// TwinCAT 3 PLC project Name
// ProgramVersion: 3.1.4026.17
// CompilerDefines: VISU_USEPROPERTYINFO
// libraries:
//   CmpBitmapPool, * (System)
//   Tc2_Standard, * (Beckhoff Automation GmbH)
//   Tc2_System, * (Beckhoff Automation GmbH)
//   Tc2_Utilities, * (Beckhoff Automation GmbH)
//   TextListUtils, * (System)
//   VisuDialogs, * (System)
//   VisuSymbols, 4.5.0.0 (System)
// project tree:
//   DUTs/ DUT_AlarmInfo.TcDUT, DUT_ModelInfo.TcDUT, DUT_ProductData.TcDUT
//   / GlobalTextList.TcGTLO, PlcTask.TcTTO, Visualization Manager.TcVMO (not stored), VISU_TASK.TcTTO
//   GVLs/ GVL_HMI.TcGVL, GVL_Retain.TcGVL, GVL_Status.TcGVL
//   POUs/10_Station/ Station1.TcPOU
//   POUs/70_Data/ Data.TcPOU
//   POUs/80_HMI/ HMI.TcPOU
//   POUs/99_FB/ fbAlarm.TcPOU
//   POUs/ MAIN.TcPOU, Test.TcPOU
//   VISUs/ ImagePool.TcIPO (not stored), TextList.TcTLO
//   VISUs/03_SideFrame/ LowerBar.TcVIS, SideBar.TcVIS, UpperBar.TcVIS
//   VISUs/02_MainFrame/ Main.TcVIS, Data.TcVIS, Alarm.TcVIS, Setting.TcVIS, Manual.TcVIS, Model.TcVIS
//   VISUs/01_Page/ BasePage.TcVIS
// real-time tasks:
//   TASK PlcTask: cycle T#10ms, priority 6, ADS port 351
//   TASK VISU_TASK: cycle T#200000us, priority 8, ADS port 350

CONFIGURATION Name
    RESOURCE PLC ON TwinCAT3
        TASK PlcTask(INTERVAL := T#10ms, PRIORITY := 6);
        TASK VISU_TASK(INTERVAL := T#200000us, PRIORITY := 8);
        PROGRAM MAIN WITH PlcTask : MAIN;
        PROGRAM VisuElems_Visu_Prg WITH VISU_TASK : VisuElems.Visu_Prg;
    END_RESOURCE
END_CONFIGURATION

// ---- DUTs/DUT_AlarmInfo.TcDUT
TYPE DUT_AlarmInfo :
STRUCT
	bActive			: BOOL;              // 알람 활성 여부 (발생 중인지)
	iAlarmCode		: INT;               // 알람 코드 (번호)
	sAlarmMessage	: STRING(255);       // 알람 메시지 텍스트
	tTimeStamp		: DT;                // 알람 발생 시간
	sLocation		: STRING(50);         // 알람 발생 위치 (설비명 등)
	iPriority		: INT;               // 우선순위 (1:높음, 2:중간, 3:낮음 등)
END_STRUCT
END_TYPE

// ---- DUTs/DUT_ModelInfo.TcDUT
TYPE DUT_ModelInfo :
STRUCT
	iNumber		: INT;
	sName		: STRING;
	abType		: ARRAY[1..cMaxTypeNo] OF BOOL;
	aiType		: ARRAY[1..cMaxTypeNo] OF INT;
	arPosition	: ARRAY[1..cMaxPositionNo] OF LREAL;
	arSpeed		: ARRAY[1..cMaxPositionNo] OF LREAL;
END_STRUCT
END_TYPE

// ---- DUTs/DUT_ProductData.TcDUT
TYPE DUT_ProductData :
STRUCT
	sName				:STRING;				(*Product Name*)
	iType				:INT;					(*Product Name*)
	tCycleTime			:TIME;					(*Product Name*)
	tProcessTime		:TIME;					(*Product Name*)
	dtStartTime 		:DT;					(*Product Name*)
	dtEndTime			:DT;					(*Product Name*)
	iRecipeNo			:INT;					(*Product Name*)
	iInputCount			:INT;
	abInspectResult1		:BOOL;	// True = Pass (OK)
	aiInspectResultCode1	:INT;	// 0 = Pending (not inspected yet), 1 = Pass (OK), 2 = Fail – Reason #1, 3 = Fail – Reason #2
	abInspectResult2		:BOOL;	// True = Pass (OK)
	aiInspectResultCode2	:INT;	// 0 = Pending (not inspected yet), 1 = Pass (OK), 2 = Fail – Reason #1, 3 = Fail – Reason #2
	abInspectResult3		:BOOL;	// True = Pass (OK)
	aiInspectResultCode3	:INT;	// 0 = Pending (not inspected yet), 1 = Pass (OK), 2 = Fail – Reason #1, 3 = Fail – Reason #2
	abInspectResult4		:BOOL;	// True = Pass (OK)
	aiInspectResultCode4	:INT;	// 0 = Pending (not inspected yet), 1 = Pass (OK), 2 = Fail – Reason #1, 3 = Fail – Reason #2
	abInspectResult5		:BOOL;	// True = Pass (OK)
	aiInspectResultCode5	:INT;	// 0 = Pending (not inspected yet), 1 = Pass (OK), 2 = Fail – Reason #1, 3 = Fail – Reason #2
	abInspectResult6		:BOOL;	// True = Pass (OK)
	aiInspectResultCode6	:INT;	// 0 = Pending (not inspected yet), 1 = Pass (OK), 2 = Fail – Reason #1, 3 = Fail – Reason #2
END_STRUCT
END_TYPE

// ---- GVLs/GVL_HMI.TcGVL
//{attribute 'qualified_only'}
VAR_GLOBAL
	
	iSelectProductNo	: UINT; // Select Product No.
	bSaveProductData	: BOOL;
	bDeleteProductData	: BOOL;
	bDeleteRecipeData	: BOOL;
	bRemoveProductData	: BOOL;
	
// Main
	bBtAutoMode			: BOOL;
	bBtStart			: BOOL;
	bBtStop				: BOOL;
	bBtHome				: BOOL;
	bBtDoorLock			: BOOL;
	bBtDoorUnlock		: BOOL;
	bBtAlarmReset		: BOOL;
	bLpBlink			: BOOL;
	bLpHome				: BOOL;
	bLpAlarmReset		: BOOL;
	bLpAutoMode			: BOOL;
	bLpStart			: BOOL;
	
// Index
	iTextIndex			: INT;	// By 'TextList' 0= Manual, 1= Auto
	iMainFrame			: INT; // 0= Main, 1= Manual, 2= Setting, 3= Model, 4= Data, 5= Alarm

// Frame Number
    bMainScreen			: BOOL;
    bManualScreen		: BOOL;
	bSettingScreen		: BOOL;
	bModelScreen		: BOOL;
	bDataScreen			: BOOL;
	bAlarmScreen		: BOOL;
	
// Message Box
	sCurrentTitle		: STRING;
	sCurrentMessage		: STRING;
	bCallMessageBox		: BOOL;

// Time
	abStartTimeStamp	: ARRAY[0..cMaxStationNo-1] OF BOOL;
	abEndTimeStamp		: ARRAY[0..cMaxStationNo-1] OF BOOL;
	sCurrentTime		: STRING;

// Model
	iInputModelNo		: INT;
	bBtSaveModelData	: BOOL;
	bLpSaveModelData	: BOOL;
	bBtActivateModel	: BOOL;
	bLpActivateModel	: BOOL;
	bLpDiffNumber		: BOOL;
	bLpDiffName			: BOOL;
	bLpDiffbType		: BOOL;
	bLpDiffiType		: BOOL;
	bLpDiffrPosition	: BOOL;
	bLpDiffrSpeed		: BOOL;
	iModelIndex			: INT := 1;
	bInvisibleLeft		: BOOL;
	bInvisibleRight		: BOOL;

// Test Bt
	bTest				: BOOL;
END_VAR

// ---- GVLs/GVL_Retain.TcGVL
//{attribute 'qualified_only'}
 {attribute 'TcPersistent'}
VAR_GLOBAL PERSISTENT
//Product Data
	astProductData 		: ARRAY[0..cMaxStationNo+1] OF DUT_ProductData;
	abMoveShift			: ARRAY[0..cMaxStationNo] OF BOOL;

// Alarm
	astAlarmHistory		: ARRAY[0..cMaxAlarmLogCount-1] OF DUT_AlarmInfo; // 최근 100개 알람 저장

// Model
	astInputModel		: ARRAY[1..cMaxModelNo] OF dut_ModelInfo;
	astModel			: ARRAY[1..cMaxModelNo] OF dut_ModelInfo;
	stCurrnetModel		: dut_ModelInfo;	
END_VAR

VAR_GLOBAL CONSTANT
	cMaxAlarmLogCount	: INT := 100; 
	cMaxStationNo 		: INT := 30;
	cMaxTypeNo			: INT := 20;
	cMaxPositionNo		: INT := 30;
	cMaxModelNo			: INT := 10;
	cMaxStationAlarmNo	: INT := 100;
	
END_VAR

// ---- GVLs/GVL_Status.TcGVL
//{attribute 'qualified_only'}
VAR_GLOBAL
	//DataShift
		fbLocalTime 		: FB_LocalSystemTime;
		
	//Status
		bAutoMode				:BOOL;
		bManualMode				:BOOL;
		bHomeMode				:BOOL;
		bAutoBusy				:BOOL;
		bHomeBusy				:BOOL;
		bManualBusy				:BOOL;
		bAlarm					:BOOL;
		bWarning				:BOOL;
		bHomeComplete			:BOOL;
		bSafetyDoorLocked		:BOOL;
		bSafetyDoorUnlocked		:BOOL;
		bAlarmReset				: BOOL;
		
	//Command
		bStopCmd		:BOOL;
		bAutoCmd		:BOOL;
		bHomeCmd		:BOOL;
		bDoorUnlockCmd	:BOOL;
		bDoorLockCmd	:BOOL;
		
END_VAR

// ---- POUs/MAIN.TcPOU
PROGRAM MAIN
VAR
	
END_VAR

Data();
HMI();
Station1();

IF GVL_HMI.bTest THEN
	Test();	
END_IF

END_PROGRAM

// ---- POUs/70_Data/Data.TcPOU
PROGRAM Data
VAR
	i					:INT; //loop index
END_VAR

// Local Time
	GVL_Status.fbLocalTime(bEnable := TRUE);	// Current Time

//Remove Total Product Data
	IF GVL_HMI.bRemoveProductData THEN
		FOR i := 0 TO cMaxStationNo DO
			astProductData[i] := astProductData[cMaxStationNo+1];
		END_FOR;
		GVL_HMI.bRemoveProductData := FALSE;
	END_IF

//Data Shift
	FOR i := 0 TO (cMaxStationNo) DO
		IF i > 0 AND i <= cMaxStationNo THEN  // 범위 체크 추가
			IF abMoveShift[i] = TRUE THEN
				astProductData[i] := astProductData[i-1];
				astProductData[i-1] := astProductData[cMaxStationNo+1]; // Delete Data before Station
				abMoveShift[i] := FALSE;
			END_IF
			
			IF abStartTimeStamp[i] AND GVL_Status.fbLocalTime.bValid THEN
				astProductData[i].dtStartTime := SYSTEMTIME_TO_DT(GVL_Status.fbLocalTime.systemTime);
			END_IF
			IF abEndTimeStamp[i] AND GVL_Status.fbLocalTime.bValid THEN
				astProductData[i].dtEndTime := SYSTEMTIME_TO_DT(GVL_Status.fbLocalTime.systemTime);
			END_IF		
			astProductData[i].tProcessTime	:= astProductData[i].dtEndTime - astProductData[i].dtStartTime;
		END_IF
	END_FOR;

END_PROGRAM

// ---- POUs/80_HMI/HMI.TcPOU
PROGRAM HMI
VAR
	tonBlink : ton;
	tonAlarmReset : ton;
	i	: INT;
	iDiffReset: INT;
	triModelSet: R_TRIG;
END_VAR

// Current Time
	GVL_HMI.sCurrentTime := SYSTEMTIME_TO_STRING( GVL_Status.fbLocalTime.systemTime);

// Select Auto Mode
	IF GVL_Status.bAutoCmd = FALSE AND GVL_Status.bAutoBusy = FALSE AND GVL_Status.bManualBusy = FALSE AND GVL_Status.bHomeBusy = FALSE  THEN
		//Turn On Auto Mode 
        IF GVL_HMI.bBtAutoMode = TRUE AND GVL_Status.bAutoMode = FALSE AND GVL_Status.bSafetyDoorLocked THEN
			GVL_Status.bAutoMode := TRUE;
			GVL_HMI.bBtAutoMode := FALSE;
		END_IF
		//Turn Off Auto Mode
		IF GVL_HMI.bBtAutoMode = TRUE AND GVL_Status.bAutoMode = TRUE  THEN
			GVL_Status.bAutoMode := FALSE;
			GVL_HMI.bBtAutoMode := FALSE;
		END_IF
	ELSE
		GVL_HMI.bBtAutoMode := FALSE;
	END_IF
		
        IF GVL_Status.bSafetyDoorUnlocked OR (NOT bDoorUnlockCmd AND NOT bDoorLockCmd)  THEN
		GVL_HMI.bBtAutoMode := FALSE;
	END_IF
	
	gvl_hmi.bLpAutoMode := GVL_Status.bAutoMode OR ( GVL_HMI.bLpBlink AND GVL_Status.bHomeComplete AND GVL_Status.bHomeMode);
	
// Select Manual Mode
	IF GVL_Status.bAutoMode = FALSE THEN
		GVL_Status.bManualMode := TRUE;
		GVL_HMI.iTextIndex := 0;
	ELSE
		GVL_Status.bManualMode := FALSE;
		GVL_HMI.iTextIndex := 1;
	END_IF
	
// Auto Running
	IF GVL_HMI.bBtStart = TRUE AND GVL_Status.bAutoMode = TRUE AND GVL_Status.bHomeComplete = TRUE AND GVL_Status.bAutoBusy = FALSE AND GVL_Status.bManualBusy = FALSE AND GVL_Status.bHomeBusy = FALSE THEN
		GVL_Status.bAutoCmd := TRUE;
		GVL_HMI.bBtStart := FALSE;
	ELSIF GVL_HMI.bBtStart = TRUE AND GVL_Status.bAutoMode = FALSE THEN
		GVL_HMI.bBtStart := FALSE;
	END_IF
	
	gvl_hmi.bLpStart := GVL_Status.bAutoCmd OR ( GVL_HMI.bLpBlink AND GVL_Status.bHomeComplete AND GVL_Status.bAutoMode AND ( NOT gvl_status.bAlarm AND NOT gvl_status.bWarning));
	
	
// Stop 
	IF GVL_HMI.bBtStop = TRUE AND GVL_Status.bStopCmd = FALSE THEN
		GVL_Status.bStopCmd	:= TRUE;
		GVL_HMI.bBtStop := FALSE;
	END_IF
	
	IF GVL_Status.bStopCmd = TRUE AND GVL_Status.bAutoBusy = FALSE AND GVL_Status.bManualBusy = FALSE AND GVL_Status.bHomeBusy = FALSE THEN
		GVL_Status.bAutoCmd := FALSE;
		GVL_Status.bHomeCmd := FALSE;
		GVL_Status.bStopCmd := FALSE;
		GVL_HMI.bBtStop := FALSE;
	END_IF
	
// Home 
	GVL_Status.bHomeMode := GVL_Status.bSafetyDoorLocked AND GVL_Status.bManualMode;
	
	IF GVL_HMI.bBtHome = TRUE AND GVL_Status.bHomeMode = TRUE AND GVL_Status.bAutoBusy = FALSE AND GVL_Status.bManualBusy = FALSE AND GVL_Status.bHomeBusy = FALSE AND GVL_Status.bAutoCmd = FALSE THEN
		GVL_Status.bHomeCmd := TRUE;
		GVL_HMI.bBtHome := FALSE;
	ELSIF GVL_HMI.bBtHome = TRUE AND GVL_Status.bHomeMode = FALSE THEN
		GVL_HMI.bBtHome := FALSE;
	END_IF
	
	IF GVL_Status.bHomeCmd = TRUE AND GVL_Status.bHomeComplete = TRUE THEN
		GVL_Status.bHomeCmd := FALSE;
	END_IF
	
	// bHomeComplete Reset
		IF GVL_Status.bSafetyDoorUnlocked THEN
			GVL_Status.bHomeComplete := FALSE;
		END_IF
	
		GVL_HMI.bLpHome := GVL_Status.bHomeComplete OR ( NOT GVL_Status.bHomeComplete AND GVL_Status.bHomeMode AND GVL_HMI.bLpBlink);
	
// Door Unlock
	IF GVL_HMI.bBtDoorUnlock AND GVL_Status.bManualMode AND NOT GVL_Status.bManualBusy THEN
		GVL_Status.bDoorUnlockCmd := TRUE;
		GVL_Status.bDoorLockCmd := FALSE;
		GVL_HMI.bBtDoorUnlock := FALSE;
	ELSE
		GVL_HMI.bBtDoorUnlock := FALSE;
	END_IF
	
// Door Lock
	IF GVL_HMI.bBtDoorLock AND GVL_Status.bManualMode AND NOT GVL_Status.bManualBusy THEN
		GVL_Status.bDoorLockCmd := TRUE;
		GVL_Status.bDoorUnlockCmd := FALSE;
		GVL_HMI.bBtDoorLock := FALSE;
	ELSE
		GVL_HMI.bBtDoorLock := FALSE;
	END_IF
	
// Alarm Reset
	IF gvl_hmi.bBtAlarmReset THEN
		GVL_Status.bAlarmReset := TRUE;
		gvl_hmi.bBtAlarmReset := FALSE;
	END_IF
	
	tonAlarmReset(in := GVL_Status.bAlarmReset, pt := T#0.5S);
	
	IF tonAlarmReset.Q THEN
		GVL_Status.bAlarmReset := FALSE;
	END_IF
	
	gvl_hmi.bLpAlarmReset := GVL_Status.bAlarmReset OR (GVL_HMI.bLpBlink AND (gvl_status.bAlarm OR gvl_status.bWarning));
		
// blink
 	tonBlink(in := NOT tonBlink.q , PT := T#500MS);
	
	IF tonBlink.Q THEN
		GVL_HMI.bLpBlink := NOT GVL_HMI.bLpBlink;
	END_IF
	
// Current Screen
	gvl_hmi.bMainScreen := gvl_hmi.iMainFrame = 0;
	gvl_hmi.bManualScreen := gvl_hmi.iMainFrame = 1;
	gvl_hmi.bSettingScreen := gvl_hmi.iMainFrame = 2;
	gvl_hmi.bModelScreen := gvl_hmi.iMainFrame = 3;
	gvl_hmi.bDataScreen := gvl_hmi.iMainFrame = 4;
	gvl_hmi.bAlarmScreen := gvl_hmi.iMainFrame = 5;
	
	
// Model
	 IF bModelScreen THEN
		 FOR i := 1 TO cMaxModelNo DO
			astInputModel[i].iNumber := i;
			IF bBtSaveModelData THEN
				astModel[iModelindex] := astInputModel[iModelindex];
			END_IF
			IF bBtActivateModel THEN
				 stCurrnetModel := astModel[iModelindex];
			END_IF
		 END_FOR
		 iModelindex := LIMIT(1,iModelindex,cMaxModelNo);
		 bLpDiffNumber := astInputModel[iModelindex].iNumber <> astModel[iModelindex].iNumber;
		 bLpDiffName := astInputModel[iModelindex].sName <> astModel[iModelindex].sName;
		 FOR i := 1 TO cMaxTypeNo DO
			 IF astInputModel[iModelindex].abType[i] <> astModel[iModelindex].abType[i] THEN
			 bLpDiffbType := TRUE;
			 END_IF
		 END_FOR
		 FOR i := 1 TO cMaxTypeNo DO
			 IF astInputModel[iModelindex].aiType[i] <> astModel[iModelindex].aiType[i] THEN
			 bLpDiffiType := TRUE;
			 END_IF
		 END_FOR
		 FOR i := 1 TO cMaxPositionNo DO
			 IF astInputModel[iModelindex].arPosition[i] <> astModel[iModelindex].arPosition[i] THEN
			 bLpDiffrPosition := TRUE;
			 END_IF
		 END_FOR
		 FOR i := 1 TO cMaxPositionNo DO
			 IF astInputModel[iModelindex].arSpeed[i] <> astModel[iModelindex].arSpeed[i] THEN
			 bLpDiffrSpeed := TRUE;
			 END_IF
		 END_FOR		
		 IF (iModelindex <> iDiffReset) OR bBtSaveModelData OR triModelSet.Q THEN
			 bLpDiffbType := FALSE;
			 bLpDiffiType := FALSE;
			 bLpDiffrPosition := FALSE;
			 bLpDiffrSpeed := FALSE;
			 iDiffReset := iModelindex;
		 END_IF
		 bLpSaveModelData := bBtSaveModelData OR ((bLpDiffNumber OR bLpDiffName OR bLpDiffbType OR bLpDiffiType OR bLpDiffrPosition OR bLpDiffrSpeed) AND bLpBlink);
		 bInvisibleLeft := iModelindex = 1;
		 bInvisibleRight := iModelindex = cMaxModelNo;
		 bLpActivateModel := ((NOT bLpSaveModelData AND (stCurrnetModel.iNumber = 0)) AND bLpBlink) OR bBtActivateModel;
	 END_IF
	 triModelSet(CLK:= bModelScreen, Q=> );
	 IF triModelSet.Q THEN
		 FOR i := 1 TO cMaxModelNo DO
			astInputModel[i] := astModel[i];
		 END_FOR
	 END_IF

END_PROGRAM

// ---- POUs/10_Station/Station1.TcPOU
PROGRAM Station1
VAR

END_VAR

END_PROGRAM

// ---- POUs/Test.TcPOU
PROGRAM Test
VAR

	fbTestAlarm1: fbalarm;

        bTestSelectWarning: BOOL;
        bTestAlarmCondition: BOOL;
	bTestError1: BOOL;
	bTestWarning1: BOOL;
	

END_VAR

// Door		
	GVL_Status.bSafetyDoorLocked := GVL_Status.bDoorLockCmd;
	GVL_Status.bSafetyDoorUnlocked := GVL_Status.bDoorUnlockCmd;
	
// home
	IF GVL_Status.bHomeCmd THEN
		GVL_Status.bHomeComplete := TRUE;
	END_IF



// Alarm
	fbTestAlarm1(
        bSelectWarning:= bTestSelectWarning,
	tDelayTime:= T#1S, 
	bCommand:= TRUE, 
        bAlarmCondition:= bTestAlarmCondition,
	iAlarmCode:= 1, 
	iPriority:= 1, 
	sAlarmMessage:= 'hello', 
	sLocation:= 'office', 
	bError=> bTestError1, 
	bWarning=> bTestWarning1);

END_PROGRAM

// ---- POUs/99_FB/fbAlarm.TcPOU
FUNCTION_BLOCK fbAlarm	// 
VAR_INPUT
	bSelectWarning	: BOOL;
	tDelayTime	: TIME;
	bCommand	: BOOL;
	bAlarmCondition	: BOOL;
	iAlarmCode	: INT;
	iPriority	: INT;
	sAlarmMessage	: STRING;
	sLocation	: STRING;
END_VAR
VAR_OUTPUT
	bError	: BOOL;
	bWarning	: BOOL;
END_VAR
VAR
	bAlarm	: BOOL;
	triAlarm	: R_Trig;
	triWarning	: R_Trig;
	triError	: R_Trig;
	i: INT;
	stAlarmInfo	: Dut_AlarmInfo;
	tonDelayTimer	: ton;
END_VAR


// Alarm Input
	bAlarm	:= bCommand AND bAlarmCondition;
	tonDelayTimer(in := bAlarm, pt :=tDelayTime);

// Alarm History
	triAlarm(clk := tonDelayTimer.Q);
	IF triAlarm.Q THEN
		FOR i := cMaxAlarmLogCount TO 1 BY -1 DO
			astAlarmHistory[i]	:= astAlarmHistory[i-1];
		END_FOR
		stAlarmInfo.iAlarmCode	:= iAlarmCode;
		stAlarmInfo.iPriority	:= iPriority;
		stAlarmInfo.sAlarmMessage	:= sAlarmMessage;
		stAlarmInfo.sLocation	:= sLocation;
		stAlarmInfo.tTimeStamp	:= SYSTEMTIME_TO_DT(GVL_Status.fbLocalTime.systemTime);
		astAlarmHistory[0] := stAlarmInfo;
	END_IF

// Alarm Output
	IF tonDelayTimer.Q THEN
		bError := NOT bSelectWarning;
		gvl_status.bAlarm := NOT bSelectWarning;
		bWarning := bSelectWarning;
		gvl_status.bWarning := bSelectWarning;
	END_IF
	
// Alarm Reset
	IF bAlarmReset THEN
		bError := FALSE;
		bWarning := FALSE;
		gvl_status.bAlarm := FALSE;
		gvl_status.bWarning := FALSE;
	END_IF
	
// Call Message Box
	triWarning(clk := gvl_status.bWarning);
	IF triWarning.Q THEN
		sCurrentTitle	:= astAlarmHistory[0].sLocation;
		sCurrentMessage	:= astAlarmHistory[0].sAlarmMessage;
		bCallMessageBox := gvl_status.bWarning;
	END_IF
	
// Change Main Frame to Alarm
	triError(clk := gvl_status.bAlarm);
	IF triError.Q THEN
		iMainFrame := 5;
	END_IF

END_FUNCTION_BLOCK

// ---- GlobalTextList.TcGTLO
TEXTLIST GlobalTextList
  422 = '%.19s' | Korea: '%.19s' | English: '%.19s'
  792 = '%i'
  75 = '%s'
  500 = '1'
  410 = 'a'
  336 = 'Activate Model'
  479 = 'Activate Name : %s'
  578 = 'Activate No : %i'
  851 = 'Active'
  609 = 'Alarm'
  662 = 'Alarm Code'
  947 = 'Alarm Page'
  35 = 'Alarm Reset'
  411 = 'AlarmCode'
  22 = 'AlarmMessage'
  147 = 'AlarmReset' | Korea: '초기화'
  23 = 'Alarm_Log'
  557 = 'Arkplus' | Korea: '화면인터페이스' | English: 'Standard_HMI'
  984 = 'Assemble1'
  741 = 'Assemble2'
  530 = 'Assemble3'
  491 = 'Auto Mode'
  808 = 'AutoMode'
  787 = 'b'
  699 = 'Code'
  709 = 'Conveyor'
  734 = 'Conveyor Pitch'
  977 = 'Current %s'
  122 = 'Data'
  161 = 'Data Page'
  928 = 'dfasdffffffffffffffffffffffffffffff'
  215 = 'Disable'
  226 = 'Door'
  850 = 'Door Close'
  103 = 'Door Open'
  567 = 'DoorClose'
  32 = 'Enable'
  271 = 'English' | Korea: '영어' | English: 'English'
  697 = 'fdsafdafsda'
  217 = 'GroupBox'
  279 = 'Home'
  993 = 'Inspection1'
  456 = 'Inspection2'
  921 = 'Inspection3'
  332 = 'Korea' | Korea: '한국어' | English: 'Korea'
  0 = 'Location'
  956 = 'Main'
  707 = 'Main Page'
  301 = 'Manual'
  775 = 'Manual Page'
  83 = 'ManualMode'
  186 = 'Message'
  376 = 'Model'
  601 = 'Model Name %s'
  313 = 'Model Page'
  136 = 'Name'
  599 = 'Name %s'
  828 = 'No : %i'
  259 = 'No : %s'
  536 = 'Parameter'
  975 = 'Pos %5.2f'
  395 = 'Pos %d'
  403 = 'Priority'
  529 = 'Robot'
  204 = 'SafetyBypass'
  331 = 'Sample'
  908 = 'Save Model'
  239 = 'Setting'
  394 = 'Setting Page'
  181 = 'Spd %5.2f'
  125 = 'Speed'
  849 = 'Standard_HMI' | Korea: '화면인터페이스'
  261 = 'Start'
  606 = 'Stop'
  904 = 'Test'
  272 = 'Time Stamp'
  199 = 'TimeStamp'
  396 = 'TurnTable'
  712 = 'type'
  334 = 'Type01'
  446 = 'Type02'
  966 = 'Type03'
  706 = 'Type04'
  126 = 'Type05'
  809 = 'Type06'
  245 = 'Type07'
  162 = 'Type08'
  992 = 'Type09'
  710 = 'Type10'
  26 = 'Unit1 Assemble'
  926 = 'Unit1 End'
  600 = 'Unit1 Position1'
  943 = 'Unit1 Start'
  540 = 'Unit2 Position1'
  942 = 'Unit2 Start'
  16 = 'Unit3 Assemble'
  358 = 'Unit3 End'
  93 = 'Vision'
  773 = 'Vision1'
  925 = 'Vision2'
  185 = 'Vision3'
  171 = 'yyyy‑MM‑dd\xa0HH:mm:ss'
END_TEXTLIST

// ---- VISUs/03_SideFrame/LowerBar.TcVIS
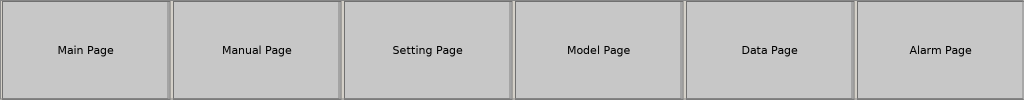
VISUALIZATION LowerBar  // 1024x100
    Button (2,1 168x99), "Main Page", colour toggle: gvl_hmi.bMainScreen
        OnMouseClick: execute { gvl_hmi.iMainFrame := 0; }
    Button (173,1 168x99), "Manual Page", colour toggle: gvl_hmi.bManualScreen
        OnMouseClick: execute { gvl_hmi.iMainFrame := 1; }
    Button (344,1 168x99), "Setting Page", colour toggle: gvl_hmi.bSettingScreen
        OnMouseClick: execute { gvl_hmi.iMainFrame := 2; }
    Button (515,1 168x99), "Model Page", colour toggle: gvl_hmi.bModelScreen
        OnMouseClick: execute { gvl_hmi.iMainFrame := 3; }
    Button (686,1 168x99), "Data Page", colour toggle: gvl_hmi.bDataScreen
        OnMouseClick: execute { gvl_hmi.iMainFrame := 4; }
    Button (857,1 168x99), "Alarm Page", colour toggle: gvl_hmi.bAlarmScreen
        OnMouseClick: execute { gvl_hmi.iMainFrame := 5; }
END_VISUALIZATION

// ---- VISUs/03_SideFrame/SideBar.TcVIS
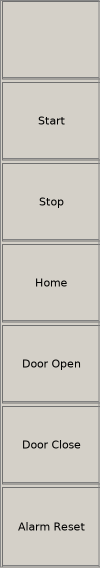
VISUALIZATION SideBar  // 100x568
    Button (2,1 99x78), colour toggle: GVL_HMI.bLpAutoMode, text list: 'TextList', text index: GVL_HMI.iTextIndex
        OnMouseClick: execute { GVL_HMI.bBtAutoMode := true; }
    Button (2,82 99x78), "Start", colour toggle: gvl_hmi.bLpStart
        OnMouseClick: execute { GVL_HMI.bBtStart := TRUE; }
    Button (2,163 99x78), "Stop", colour toggle: GVL_Status.bStopCmd
        OnMouseClick: execute { GVL_HMI.bBtStop := True; }
    Button (2,244 99x78), "Home", colour toggle: GVL_HMI.bLpHome
        OnMouseClick: execute { GVL_HMI.bBtHome := True; }
    Button (2,325 99x78), "Door Open", colour toggle: GVL_Status.bSafetyDoorUnlocked
        OnMouseClick: execute { GVL_HMI.bBtDoorUnlock := True; }
    Button (2,406 99x78), "Door Close", colour toggle: GVL_Status.bSafetyDoorLocked
        OnMouseClick: execute { GVL_HMI.bBtDoorLock := True; }
    Button (2,487 99x80), "Alarm Reset", colour toggle: gvl_hmi.bLpAlarmReset
        OnMouseClick: execute { GVL_HMI.bBtAlarmReset := True; }
END_VISUALIZATION

// ---- VISUs/03_SideFrame/UpperBar.TcVIS
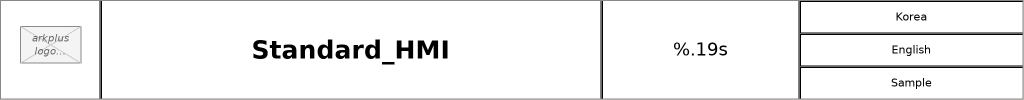
VISUALIZATION UpperBar  // 1024x100
    Rectangle (0,0 100x99)
    Image (20,26 61x37), image: arkplus logo_Resize
    Rectangle (101,0 500x99), "Standard_HMI"
    Rectangle (602,0 197x99), "%.19s", text variable: GVL_HMI.sCurrentTime
    Rectangle (800,1 223x32), "Korea"
        OnMouseClick: ChangeLanguage ChangeLanguage=Korea
    Rectangle (800,34 223x32), "English"
        OnMouseClick: ChangeLanguage ChangeLanguage=English
    Rectangle (800,67 223x32), "Sample"
END_VISUALIZATION

// ---- VISUs/02_MainFrame/Main.TcVIS
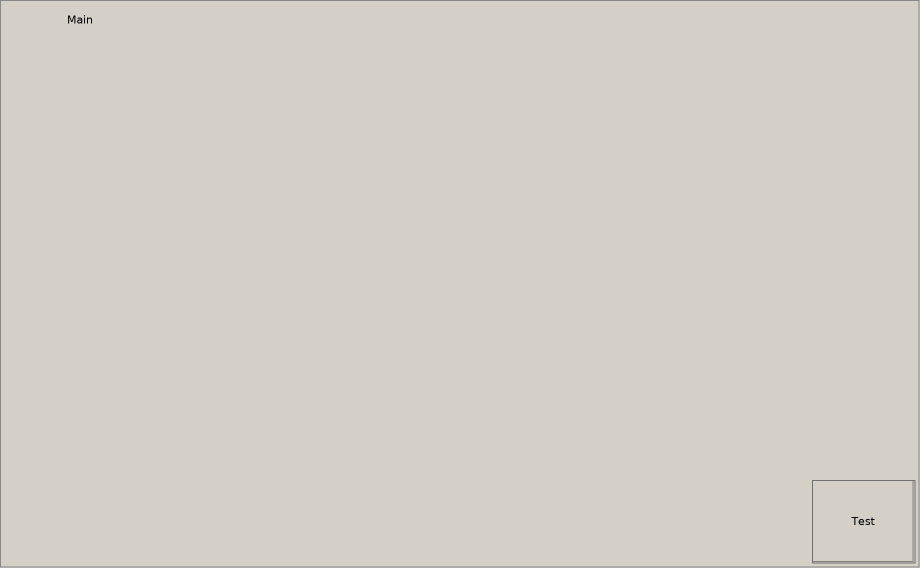
VISUALIZATION Main  // 920x568
    Label (5,5 150x30), "Main"
    Button (812,480 103x83), "Test", colour toggle: GVL_HMI.bTest
        toggle GVL_HMI.bTest
END_VISUALIZATION

// ---- VISUs/02_MainFrame/Data.TcVIS
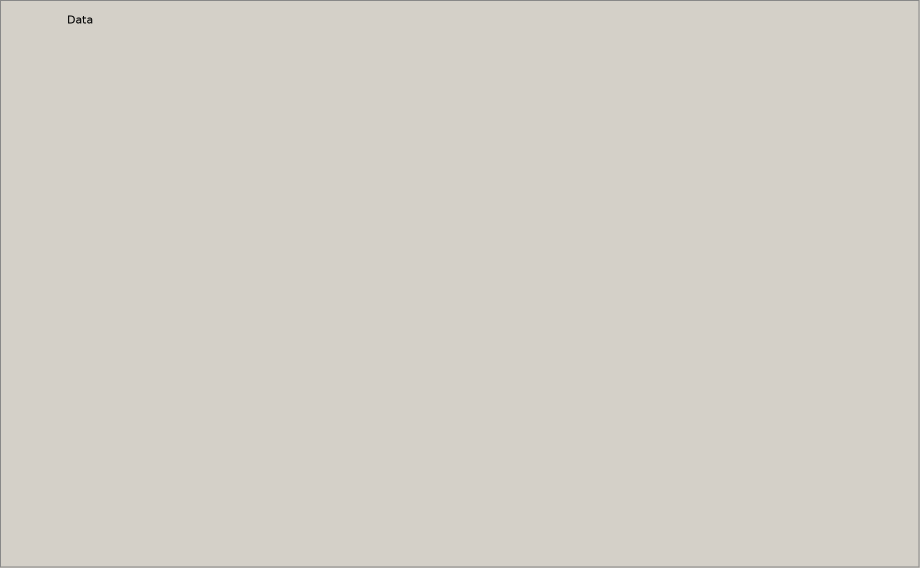
VISUALIZATION Data  // 920x568
    Label (5,5 150x30), "Data"
END_VISUALIZATION

// ---- VISUs/02_MainFrame/Alarm.TcVIS
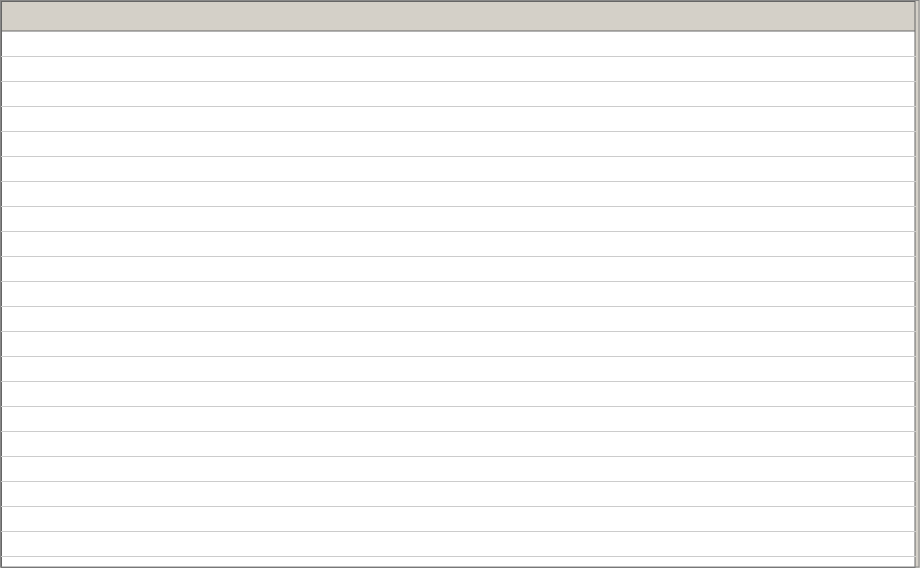
VISUALIZATION Alarm  // 920x568
    Table (1,1 914x567), data array: GVL_Retain.astAlarmHistory
        p3854506369: GVL_Retain.astAlarmHistory[INDEX].bActive
        p1892666644: GVL_Retain.astAlarmHistory[INDEX].iAlarmCode
        p338671338: GVL_Retain.astAlarmHistory[INDEX].sAlarmMessage
        p2170511999: GVL_Retain.astAlarmHistory[INDEX].tTimeStamp
        p3723444502: GVL_Retain.astAlarmHistory[INDEX].sLocation
        p1218418051: GVL_Retain.astAlarmHistory[INDEX].iPriority
        p4092479075: Time Stamp
        p1014161805: 99 - 0 + INT#1
        p1128707560: cMaxAlarmLogCount
END_VISUALIZATION

// ---- VISUs/02_MainFrame/Setting.TcVIS
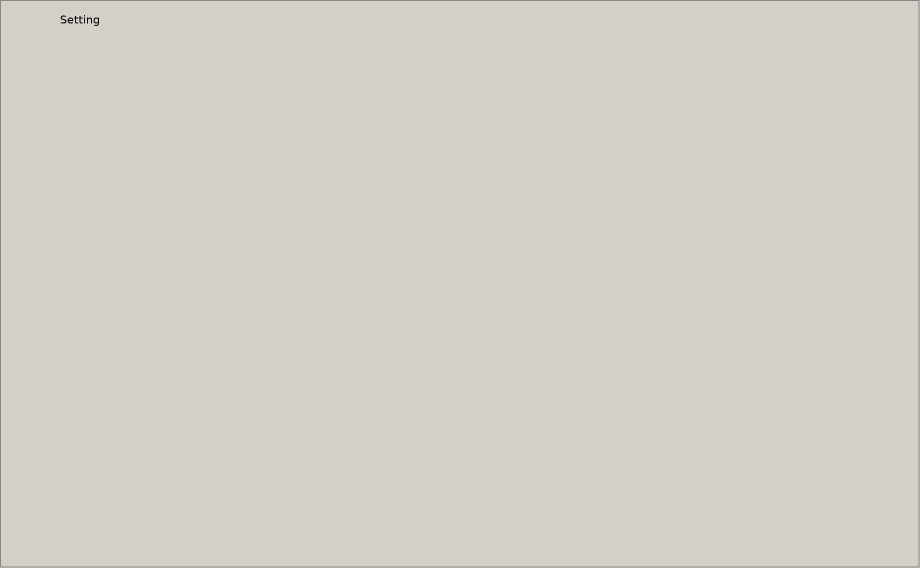
VISUALIZATION Setting  // 920x568
    Label (5,5 150x30), "Setting"
END_VISUALIZATION

// ---- VISUs/02_MainFrame/Manual.TcVIS
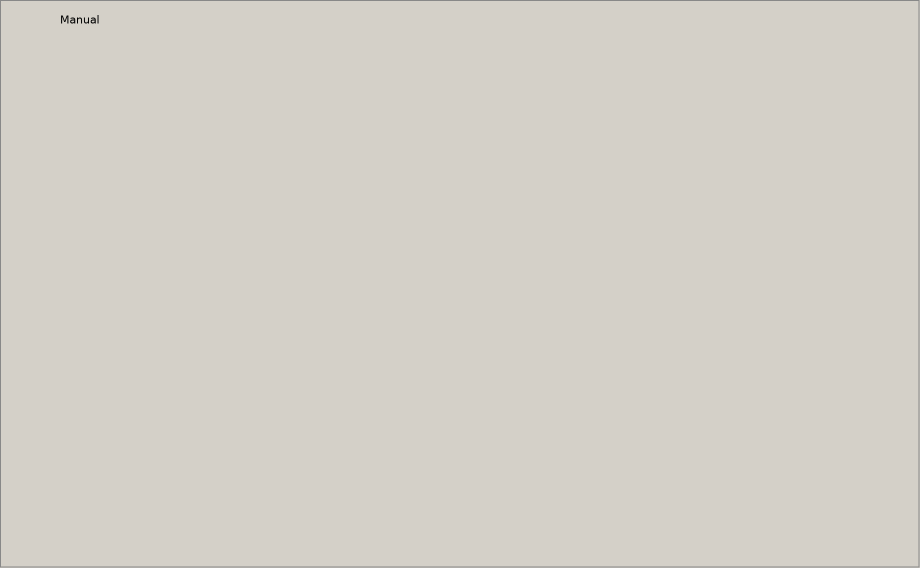
VISUALIZATION Manual  // 920x568
    Label (5,5 150x30), "Manual"
END_VISUALIZATION

// ---- VISUs/02_MainFrame/Model.TcVIS
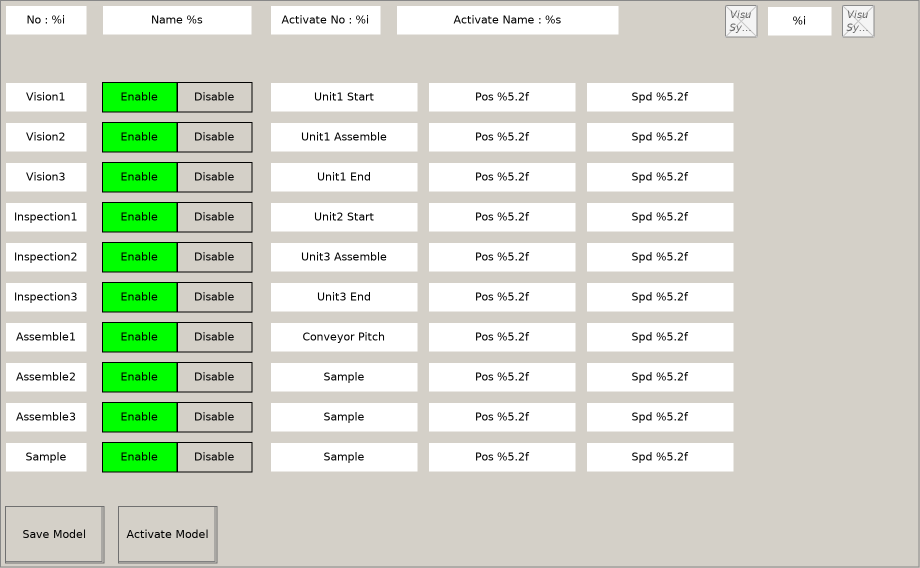
VISUALIZATION Model  // 920x568
    Textfield (102,5 150x30), "Name %s", text variable: astInputModel[iModelIndex].sName
        OnMouseClick: write the text variable via Edit
    Textfield (5,5 82x30), "No : %i", text variable: astInputModel[iModelIndex].iNumber
    Image (725,5 32x32), invisible if: bInvisibleLeft, image: VisuSymbols.Symbols.ArrowBoldLeft
        OnMouseClick: execute { iModelindex := iModelindex -1; }
    Image (842,5 32x32), invisible if: bInvisibleRight, image: VisuSymbols.Symbols.ArrowBoldRight
        OnMouseClick: execute { iModelindex := iModelindex +1; }
    Textfield (767,6 65x30), "%i", text variable: astInputModel[iModelIndex].iNumber
        OnMouseClick: write iModelIndex via Default, min 1, max cMaxModelNo
    Textfield (5,82 82x30), "Vision1"
    Rectangle (102,82 75x30), "Enable", colour toggle: astInputModel[iModelIndex].abType[1]
        OnMouseClick: execute { astInputModel[iModelIndex].abType[1] := FALSE; }
    Rectangle (177,82 75x30), "Disable", colour toggle: astInputModel[iModelIndex].abType[1]
        OnMouseClick: execute { astInputModel[iModelIndex].abType[1] := true; }
    Textfield (5,122 82x30), "Vision2"
    Rectangle (102,122 75x30), "Enable", colour toggle: astInputModel[iModelIndex].abType[2]
        OnMouseClick: execute { astInputModel[iModelIndex].abType[2] := FALSE; }
    Rectangle (177,122 75x30), "Disable", colour toggle: astInputModel[iModelIndex].abType[2]
        OnMouseClick: execute { astInputModel[iModelIndex].abType[2] := true; }
    Textfield (5,162 82x30), "Vision3"
    Rectangle (102,162 75x30), "Enable", colour toggle: astInputModel[iModelIndex].abType[3]
        OnMouseClick: execute { astInputModel[iModelIndex].abType[3] := FALSE; }
    Rectangle (177,162 75x30), "Disable", colour toggle: astInputModel[iModelIndex].abType[3]
        OnMouseClick: execute { astInputModel[iModelIndex].abType[3] := true; }
    Textfield (5,202 82x30), "Inspection1"
    Rectangle (102,202 75x30), "Enable", colour toggle: astInputModel[iModelIndex].abType[4]
        OnMouseClick: execute { astInputModel[iModelIndex].abType[4] := FALSE; }
    Rectangle (177,202 75x30), "Disable", colour toggle: astInputModel[iModelIndex].abType[4]
        OnMouseClick: execute { astInputModel[iModelIndex].abType[4] := true; }
    Textfield (5,242 82x30), "Inspection2"
    Rectangle (102,242 75x30), "Enable", colour toggle: astInputModel[iModelIndex].abType[5]
        OnMouseClick: execute { astInputModel[iModelIndex].abType[5] := FALSE; }
    Rectangle (177,242 75x30), "Disable", colour toggle: astInputModel[iModelIndex].abType[5]
        OnMouseClick: execute { astInputModel[iModelIndex].abType[5] := true; }
    Textfield (5,282 82x30), "Inspection3"
    Rectangle (102,282 75x30), "Enable", colour toggle: astInputModel[iModelIndex].abType[6]
        OnMouseClick: execute { astInputModel[iModelIndex].abType[6] := FALSE; }
    Rectangle (177,282 75x30), "Disable", colour toggle: astInputModel[iModelIndex].abType[6]
        OnMouseClick: execute { astInputModel[iModelIndex].abType[6] := true; }
    Textfield (5,322 82x30), "Assemble1"
    Rectangle (102,322 75x30), "Enable", colour toggle: astInputModel[iModelIndex].abType[7]
        OnMouseClick: execute { astInputModel[iModelIndex].abType[7] := FALSE; }
    Rectangle (177,322 75x30), "Disable", colour toggle: astInputModel[iModelIndex].abType[7]
        OnMouseClick: execute { astInputModel[iModelIndex].abType[7] := true; }
    Textfield (5,362 82x30), "Assemble2"
    Rectangle (102,362 75x30), "Enable", colour toggle: astInputModel[iModelIndex].abType[8]
        OnMouseClick: execute { astInputModel[iModelIndex].abType[8] := FALSE; }
    Rectangle (177,362 75x30), "Disable", colour toggle: astInputModel[iModelIndex].abType[8]
        OnMouseClick: execute { astInputModel[iModelIndex].abType[8] := true; }
    Textfield (5,402 82x30), "Assemble3"
    Rectangle (102,402 75x30), "Enable", colour toggle: astInputModel[iModelIndex].abType[9]
        OnMouseClick: execute { astInputModel[iModelIndex].abType[9] := FALSE; }
    Rectangle (177,402 75x30), "Disable", colour toggle: astInputModel[iModelIndex].abType[9]
        OnMouseClick: execute { astInputModel[iModelIndex].abType[9] := true; }
    Textfield (5,442 82x30), "Sample"
    Rectangle (102,442 75x30), "Enable", colour toggle: astInputModel[iModelIndex].abType[10]
        OnMouseClick: execute { astInputModel[iModelIndex].abType[10] := FALSE; }
    Rectangle (177,442 75x30), "Disable", colour toggle: astInputModel[iModelIndex].abType[10]
        OnMouseClick: execute { astInputModel[iModelIndex].abType[10] := true; }
    Button (5,506 99x57), "Save Model", colour toggle: bLpSaveModelData
        tap bBtSaveModelData
    Button (118,506 99x57), "Activate Model", colour toggle: bLpActivateModel
        tap bBtActivateModel
    Textfield (396,5 223x30), "Activate Name : %s", text variable: stCurrnetModel.sName
        OnMouseClick: write the text variable via Edit
    Textfield (270,5 111x30), "Activate No : %i", text variable: stCurrnetModel.iNumber
    Group (270,82 148x390)
        Textfield (0,0 148x30), "Unit1 Start"
        Textfield (0,40 148x30), "Unit1 Assemble"
        Textfield (0,80 148x30), "Unit1 End"
        Textfield (0,120 148x30), "Unit2 Start"
        Textfield (0,160 148x30), "Unit3 Assemble"
        Textfield (0,200 148x30), "Unit3 End"
        Textfield (0,240 148x30), "Conveyor Pitch"
        Textfield (0,280 148x30), "Sample"
        Textfield (0,320 148x30), "Sample"
        Textfield (0,360 148x30), "Sample"
    Textfield (428,82 148x30), "Pos %5.2f", text variable: astInputModel[iModelindex].arPosition[1]
        OnMouseClick: write the text variable via Default
    Textfield (428,122 148x30), "Pos %5.2f", text variable: astInputModel[iModelindex].arPosition[2]
        OnMouseClick: write the text variable via Default
    Textfield (428,162 148x30), "Pos %5.2f", text variable: astInputModel[iModelindex].arPosition[3]
        OnMouseClick: write the text variable via Default
    Textfield (428,202 148x30), "Pos %5.2f", text variable: astInputModel[iModelindex].arPosition[4]
        OnMouseClick: write the text variable via Default
    Textfield (428,242 148x30), "Pos %5.2f", text variable: astInputModel[iModelindex].arPosition[5]
        OnMouseClick: write the text variable via Default
    Textfield (428,282 148x30), "Pos %5.2f", text variable: astInputModel[iModelindex].arPosition[6]
        OnMouseClick: write the text variable via Default
    Textfield (428,322 148x30), "Pos %5.2f", text variable: astInputModel[iModelindex].arPosition[7]
        OnMouseClick: write the text variable via Default
    Textfield (428,362 148x30), "Pos %5.2f", text variable: astInputModel[iModelindex].arPosition[8]
        OnMouseClick: write the text variable via Default
    Textfield (428,402 148x30), "Pos %5.2f", text variable: astInputModel[iModelindex].arPosition[9]
        OnMouseClick: write the text variable via Default
    Textfield (428,442 148x30), "Pos %5.2f", text variable: astInputModel[iModelindex].arPosition[10]
        OnMouseClick: write the text variable via Default
    Textfield (586,82 148x30), "Spd %5.2f", text variable: astInputModel[iModelindex].arSpeed[1]
        OnMouseClick: write the text variable via Default
    Textfield (586,122 148x30), "Spd %5.2f", text variable: astInputModel[iModelindex].arSpeed[2]
        OnMouseClick: write the text variable via Default
    Textfield (586,162 148x30), "Spd %5.2f", text variable: astInputModel[iModelindex].arSpeed[3]
        OnMouseClick: write the text variable via Default
    Textfield (586,202 148x30), "Spd %5.2f", text variable: astInputModel[iModelindex].arSpeed[4]
        OnMouseClick: write the text variable via Default
    Textfield (586,242 148x30), "Spd %5.2f", text variable: astInputModel[iModelindex].arSpeed[5]
        OnMouseClick: write the text variable via Default
    Textfield (586,282 148x30), "Spd %5.2f", text variable: astInputModel[iModelindex].arSpeed[6]
        OnMouseClick: write the text variable via Default
    Textfield (586,322 148x30), "Spd %5.2f", text variable: astInputModel[iModelindex].arSpeed[7]
        OnMouseClick: write the text variable via Default
    Textfield (586,362 148x30), "Spd %5.2f", text variable: astInputModel[iModelindex].arSpeed[8]
        OnMouseClick: write the text variable via Default
    Textfield (586,402 148x30), "Spd %5.2f", text variable: astInputModel[iModelindex].arSpeed[9]
        OnMouseClick: write the text variable via Default
    Textfield (586,442 148x30), "Spd %5.2f", text variable: astInputModel[iModelindex].arSpeed[10]
        OnMouseClick: write the text variable via Default
END_VISUALIZATION

// ---- VISUs/01_Page/BasePage.TcVIS
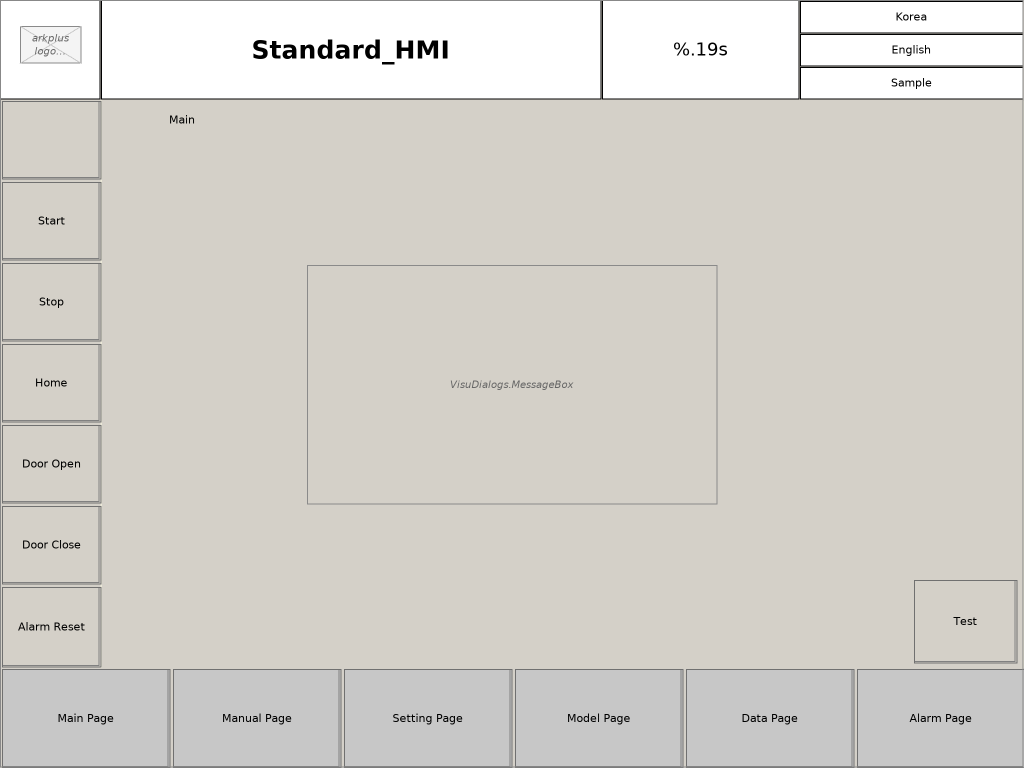
VISUALIZATION BasePage  // 1024x768
    Frame (0,0 1024x100)
        shows UpperBar()
    Frame (0,668 1024x100)
        shows LowerBar()
    Frame (0,100 100x568)
        shows SideBar()
    Frame (102,100 920x568), frame switch variable: GVL_HMI.iMainFrame
        shows Main()
        shows Manual()
        shows Setting()
        shows Model()
        shows Data()
        shows Alarm()
    Frame (307,265 410x239), invisible if: not bCallMessageBox
        shows VisuDialogs.MessageBox(eType := VisuDialogs.MessageBoxDialog_Types.OK_CANCEL, sTitle := sCurrentTitle, sMessageTxt := sCurrentMessage)
        OnMouseClick: execute { bCallMessageBox := false; }
END_VISUALIZATION

// ---- VISUs/TextList.TcTLO
TEXTLIST TextList
  0 = 'Manual' | Korea: '수동' | English: 'Manual'
  1 = 'Auto' | Korea: '자동' | English: 'Auto'
   = ''
END_TEXTLIST
